{attribute 'no_check'}
//Sequence handle object contains all needed variables for a state machine, like timer, state variable and error handle object
FUNCTION_BLOCK SEQUENCE_HDL
VAR_INPUT
	State													:	DINT := 0;		//Current state
	Err														:	ERROR_HDL;		//Error handle object
	Text													:	STRING := '';	//Could used for user defined texts 
END_VAR             										
VAR_OUTPUT          										
	MemSetState												:	DINT := 0;		//Memory for start state , set by method "Set"
	Busy													:	BOOL := FALSE;	//State machine is active - sets to TRUE by method "Set" and state <> 0
	Done													:	BOOL := FALSE;	//State machine sucessful finished - sets to TRUE by method "Finish" if Error handle is emnpty
	TON														:	TON := (IN := FALSE); //Use Methods to control state machine time
END_VAR             	
VAR                 	
END_VAR

;

METHOD PUBLIC abort : BOOL //Return value = TRUE - state will reset to 0 and Busy to FALSE in case state was <> 0 
VAR_INPUT
END_VAR
IF state <> 0 
THEN
	Busy 													:= FALSE;
	Done 													:= FALSE;
	     													  													
	text 													:= CONCAT('ABORTED~State:',DINT_TO_STRING(state));
	text 													:= CONCAT(text,'(SetState:');
	text 													:= CONCAT(text,DINT_TO_STRING(MemSetState));
	text 													:= CONCAT(text,')/Busy=');
	text 													:= CONCAT(text,BOOL_TO_STRING(Busy));
	text 													:= CONCAT(text,'/Done=');
	text 													:= CONCAT(text,BOOL_TO_STRING(Done));
	text 													:= CONCAT(text,'/Error=');
	text 													:= CONCAT(text,BOOL_TO_STRING(Err.flag));
	
	state													:= 0;
	Abort 													:= TRUE;
ELSE
	Abort 													:= TRUE;
END_IF
END_METHOD

METHOD PUBLIC active : BOOL //Return value = TRUE if sequence handle is active (state <> 0)
VAR_INPUT
END_VAR
Busy														:= State <> 0;
Done														:= FALSE;
Active														:= Busy;
END_METHOD

METHOD PUBLIC finish : BOOL//Return value = TRUE if state was <> 0 and Err.flag = FALSE
VAR_INPUT
END_VAR
IF state <> 0 
THEN
	Busy 													:= FALSE;
	Done 													:= NOT Err.flag;
	     													  													
	text 													:= CONCAT('FINISH~State:',DINT_TO_STRING(state));
	text 													:= CONCAT(text,'(SetState:');
	text 													:= CONCAT(text,DINT_TO_STRING(MemSetState));
	text 													:= CONCAT(text,')/Busy=');
	text 													:= CONCAT(text,BOOL_TO_STRING(Busy));
	text 													:= CONCAT(text,'/Done=');
	text 													:= CONCAT(text,BOOL_TO_STRING(Done));
	
	state													:= 0;
	Finish 													:= Done;	
ELSE
	Finish 													:= FALSE;
END_IF
END_METHOD

METHOD PUBLIC incState : BOOL //Increment State by NoOfIncrements / Result always true 
VAR_INPUT
	NoOfIncrements								:	DINT;
END_VAR
State := State + NoOfIncrements;
incState := TRUE;
END_METHOD

METHOD PUBLIC reset : BOOL //return value = TRUE if execution finished 
VAR_INPUT
END_VAR
Done 														:= FALSE;
Busy 														:= FALSE;
text 														:= CONCAT('RESET~State:',DINT_TO_STRING(state));
text 														:= CONCAT(text,'(SetState:');
text 														:= CONCAT(text,DINT_TO_STRING(MemSetState));
text 														:= CONCAT(text,')/Busy=');
text 														:= CONCAT(text,BOOL_TO_STRING(Busy));
text 														:= CONCAT(text,'/Done=');
text 														:= CONCAT(text,BOOL_TO_STRING(Done));

MemSetState := state 										:=  0;
reset 														:= TRUE;
END_METHOD

METHOD PUBLIC resetWithErrHdl : BOOL //return value = TRUE if execution finished 
VAR_INPUT
END_VAR
Reset();
Err.Reset();
ResetWithErrHdl												 := TRUE;
END_METHOD

METHOD PUBLIC set : BOOL //Set MemSetstate to state value, Return value = TRUE if sequence handle will be busy (State <> 0)
VAR_INPUT
	State													:		 DINT;
END_VAR
MemSetState 												:= THIS^.state := State;
Busy 														:= state <> 0;
Done 														:= FALSE;
Set															:= Busy;
                    										
text 														:= CONCAT('SET~State:',DINT_TO_STRING(MemSetstate));
END_METHOD

PROPERTY PUBLIC ton_BT : TIME
GET
IF ton.IN
	AND NOT ton.Q
THEN
	Ton_BT 													:= ton.PT - ton.ET;
ELSE       													
	Ton_BT 													:= T#0MS;
END_IF
END_GET
END_PROPERTY

PROPERTY PUBLIC ton_PT : TIME
GET
Ton_PT 														:= ton.PT;
END_GET
SET // PUBLIC
Ton.PT 														:= Ton_PT;
END_SET
END_PROPERTY

METHOD PUBLIC tonOFF : BOOL //Return value = TRUE if execution finished
VAR_INPUT
END_VAR
TON(In := FALSE,Q => );
TonOFF := NOT Ton.Q;
END_METHOD

METHOD PUBLIC tonON : BOOL; //Return value = TRUE if execution finished
VAR_INPUT
END_VAR
TON(In := TRUE,Q => TonON);
END_METHOD

METHOD PUBLIC tonRUN : BOOL //Return value status of time (Ton.Q)
VAR_INPUT
	IN														:	BOOL;
	PT														:	TIME;
END_VAR
THIS^.TON.IN := IN;
THIS^.TON.PT := PT;
TON(IN := IN , PT := PT, Q => TonRUN);
END_METHOD

END_FUNCTION_BLOCK

(* stored: Version 1.1.0.1, ProductVersion 3.1.4024.13
   POU SEQUENCE_HDL: Id {aa74b748-c768-4296-a2fc-41ba9ed57182}, SpecialFunc None
   Method abort: Id {a4eb6e7b-b0a8-416d-846d-2f44cd210519}
   Method active: Id {08f89166-34c4-4368-bcdc-3ed0c4ed6ab6}
   Method finish: Id {2874e965-38bb-4119-98e2-eba3e25ac0a2}
   Method incState: Id {4e29fa77-cf0f-4a6f-a5f2-0c96a9ede638}
   Method reset: Id {fcfcea69-4e30-4d8a-97ad-3d23847e22cc}
   Method resetWithErrHdl: Id {a296fc9e-e145-4b85-bd19-e7f196163e9e}
   Method set: Id {42bb9387-8611-49ac-8e8e-f1186f0a93c3}
   Property ton_BT: Id {c0685f15-62bd-4ec8-a34e-03a058759ea2}
   Get Get: Id {f01f93e1-12c1-4be5-9917-8a7fc952d4ec}
   Property ton_PT: Id {c3de0b17-e41e-45ea-baa1-45e46932b1a5}
   Get Get: Id {afe92ad7-02d8-4f6f-be00-13e13b26b6da}
   Set Set: Id {f2642873-ee6d-481a-972e-e816ed609ad6}
   Method tonOFF: Id {15bdd105-bfca-496f-9a98-c8a627daccaa}
   Method tonON: Id {09ca4010-695d-4533-848d-c9b1c9fe7de3}
   Method tonRUN: Id {c820356e-eda5-42d7-b973-3c056ffef969} *)
